// TIA Portal V19 export
TYPE "typeSafetyZoneStatus"
// Status of safety zone
// stored: Access Published, IsFailsafeCompliant true, Namespace Safety
   STRUCT
      safetyReleased { ExternalWritable := 'False'} : Bool;   // Safety zone is released
      ackReq { ExternalWritable := 'False'} : Bool;   // Acknowledge is required
      safetyFault { ExternalWritable := 'False'} : Bool;   // Safety fault in at least one device is active
   END_STRUCT;
END_TYPE
